// TIA Portal V20 export
FUNCTION "01 T1-A ARUNC Alarms" : Void   // FC1102, LAD
TITLE = ALARMS
{ S7_Optimized_Access := 'TRUE' }
// stored: AutoNumber false, IsIECCheckEnabled true, SetENOAutomatically false
   VAR_TEMP
      Trash : Bool;
   END_VAR
BEGIN

REGION Network 1: ============ ALARMS RESET ============
END_REGION

REGION Network 2: Alarms Reset
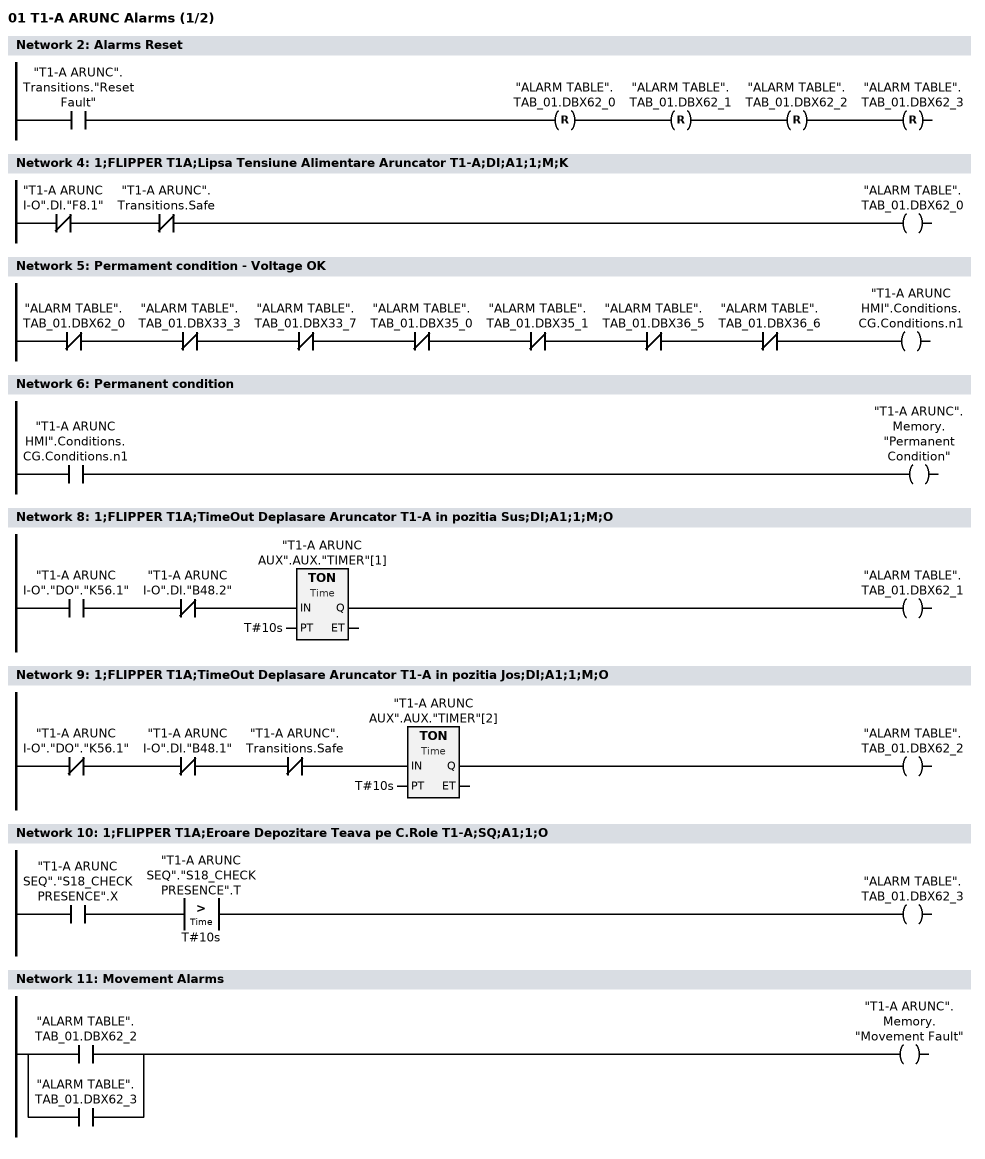
   RUNG wire#powerrail
      Contact( "T1-A ARUNC".Transitions."Reset Fault" )
      R_Coil( "ALARM TABLE".TAB_01.DBX62_0 )
      R_Coil( "ALARM TABLE".TAB_01.DBX62_1 )
      R_Coil( "ALARM TABLE".TAB_01.DBX62_2 )
      R_Coil( "ALARM TABLE".TAB_01.DBX62_3 )
   END_RUNG
   // the same network as SCL:
   IF "T1-A ARUNC".Transitions."Reset Fault" THEN
       "ALARM TABLE".TAB_01.DBX62_0 := FALSE;
       "ALARM TABLE".TAB_01.DBX62_1 := FALSE;
       "ALARM TABLE".TAB_01.DBX62_2 := FALSE;
       "ALARM TABLE".TAB_01.DBX62_3 := FALSE;
   END_IF;
END_REGION

REGION Network 3: ============ PERMANENT CONDITIONS ============
END_REGION

REGION Network 4: 1;FLIPPER T1A;Lipsa Tensiune Alimentare Aruncator T1-A;DI;A1;1;M;K
   RUNG wire#powerrail
      I_Contact( "T1-A ARUNC I-O".DI."F8.1" )
      I_Contact( "T1-A ARUNC".Transitions.Safe )
      Coil( "ALARM TABLE".TAB_01.DBX62_0 )
   END_RUNG
   // the same network as SCL:
   "ALARM TABLE".TAB_01.DBX62_0 := NOT "T1-A ARUNC I-O".DI."F8.1" AND NOT "T1-A ARUNC".Transitions.Safe;
END_REGION

REGION Network 5: Permament condition - Voltage OK
   RUNG wire#powerrail
      I_Contact( "ALARM TABLE".TAB_01.DBX62_0 )
      I_Contact( "ALARM TABLE".TAB_01.DBX33_3 )
      I_Contact( "ALARM TABLE".TAB_01.DBX33_7 )
      I_Contact( "ALARM TABLE".TAB_01.DBX35_0 )
      I_Contact( "ALARM TABLE".TAB_01.DBX35_1 )
      I_Contact( "ALARM TABLE".TAB_01.DBX36_5 )
      I_Contact( "ALARM TABLE".TAB_01.DBX36_6 )
      Coil( "T1-A ARUNC HMI".Conditions.CG.Conditions.n1 )
   END_RUNG
   // the same network as SCL:
   "T1-A ARUNC HMI".Conditions.CG.Conditions.n1 := NOT "ALARM TABLE".TAB_01.DBX62_0 AND NOT "ALARM TABLE".TAB_01.DBX33_3 AND NOT "ALARM TABLE".TAB_01.DBX33_7 AND NOT "ALARM TABLE".TAB_01.DBX35_0 AND NOT "ALARM TABLE".TAB_01.DBX35_1 AND NOT "ALARM TABLE".TAB_01.DBX36_5 AND NOT "ALARM TABLE".TAB_01.DBX36_6;
END_REGION

REGION Network 6: Permanent condition
   RUNG wire#powerrail
      Contact( "T1-A ARUNC HMI".Conditions.CG.Conditions.n1 )
      Coil( "T1-A ARUNC".Memory."Permanent Condition" )
   END_RUNG
   // the same network as SCL:
   "T1-A ARUNC".Memory."Permanent Condition" := "T1-A ARUNC HMI".Conditions.CG.Conditions.n1;
END_REGION

REGION Network 7: ======= MACHINE MOVEMENT CONTROL (SENSORS / ENCODERS / INTERLOCKS) =======
END_REGION

REGION Network 8: 1;FLIPPER T1A;TimeOut Deplasare Aruncator T1-A in pozitia Sus;DI;A1;1;M;O
   RUNG wire#powerrail
      Contact( "T1-A ARUNC I-O"."DO"."K56.1" )
      I_Contact( "T1-A ARUNC I-O".DI."B48.2" )
      { S7_Templates := "time_type := Time" } "T1-A ARUNC AUX".AUX."TIMER"[1].TON(pt := T#10s, et =>)
      Coil( "ALARM TABLE".TAB_01.DBX62_1 )
   END_RUNG
   // the same network as SCL:
   "T1-A ARUNC AUX".AUX."TIMER"[1].TON(IN := "T1-A ARUNC I-O"."DO"."K56.1" AND NOT "T1-A ARUNC I-O".DI."B48.2",
                           PT := T#10s);
   "ALARM TABLE".TAB_01.DBX62_1 := "T1-A ARUNC AUX".AUX."TIMER"[1].Q;
END_REGION

REGION Network 9: 1;FLIPPER T1A;TimeOut Deplasare Aruncator T1-A in pozitia Jos;DI;A1;1;M;O
   RUNG wire#powerrail
      I_Contact( "T1-A ARUNC I-O"."DO"."K56.1" )
      I_Contact( "T1-A ARUNC I-O".DI."B48.1" )
      I_Contact( "T1-A ARUNC".Transitions.Safe )
      { S7_Templates := "time_type := Time" } "T1-A ARUNC AUX".AUX."TIMER"[2].TON(pt := T#10s, et =>)
      Coil( "ALARM TABLE".TAB_01.DBX62_2 )
   END_RUNG
   // the same network as SCL:
   "T1-A ARUNC AUX".AUX."TIMER"[2].TON(IN := NOT "T1-A ARUNC I-O"."DO"."K56.1" AND NOT "T1-A ARUNC I-O".DI."B48.1" AND NOT "T1-A ARUNC".Transitions.Safe,
                           PT := T#10s);
   "ALARM TABLE".TAB_01.DBX62_2 := "T1-A ARUNC AUX".AUX."TIMER"[2].Q;
END_REGION

REGION Network 10: 1;FLIPPER T1A;Eroare Depozitare Teava pe C.Role T1-A;SQ;A1;1;O
   RUNG wire#powerrail
      Contact( "T1-A ARUNC SEQ"."S18_CHECK PRESENCE".X )
      { S7_Templates := "SrcType := Time" } GT_Contact(in1 := "T1-A ARUNC SEQ"."S18_CHECK PRESENCE".T, in2 := T#10s)
      Coil( "ALARM TABLE".TAB_01.DBX62_3 )
   END_RUNG
   // the same network as SCL:
   "ALARM TABLE".TAB_01.DBX62_3 := "T1-A ARUNC SEQ"."S18_CHECK PRESENCE".X AND ("T1-A ARUNC SEQ"."S18_CHECK PRESENCE".T > T#10s);
END_REGION

REGION Network 11: Movement Alarms
   RUNG wire#powerrail
      Contact( "ALARM TABLE".TAB_01.DBX62_2 )
      wire#w1
      Coil( "T1-A ARUNC".Memory."Movement Fault" )
   END_RUNG
   RUNG wire#powerrail
      Contact( "ALARM TABLE".TAB_01.DBX62_3 )
   END_RUNG wire#w1
   // the same network as SCL:
   "T1-A ARUNC".Memory."Movement Fault" := "ALARM TABLE".TAB_01.DBX62_2 OR "ALARM TABLE".TAB_01.DBX62_3;
END_REGION

REGION Network 12: ======= OTHER ALARMS =======
END_REGION

REGION Network 13: ======= FAULT =======
END_REGION

REGION Network 14: Fault Transition
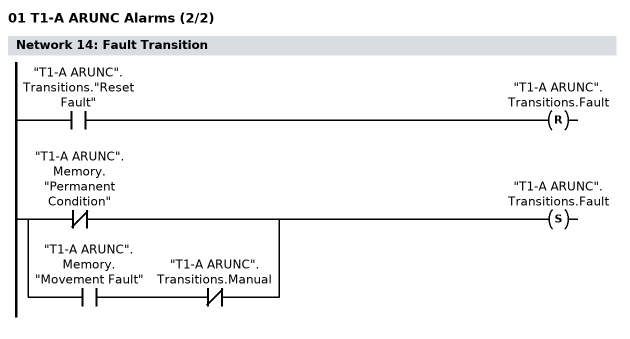
   RUNG wire#powerrail
      Contact( "T1-A ARUNC".Transitions."Reset Fault" )
      R_Coil( "T1-A ARUNC".Transitions.Fault )
   END_RUNG
   RUNG wire#powerrail
      I_Contact( "T1-A ARUNC".Memory."Permanent Condition" )
      wire#w1
      S_Coil( "T1-A ARUNC".Transitions.Fault )
   END_RUNG
   RUNG wire#powerrail
      Contact( "T1-A ARUNC".Memory."Movement Fault" )
      I_Contact( "T1-A ARUNC".Transitions.Manual )
   END_RUNG wire#w1
   // the same network as SCL:
   IF "T1-A ARUNC".Transitions."Reset Fault" THEN "T1-A ARUNC".Transitions.Fault := FALSE; END_IF;
   IF NOT "T1-A ARUNC".Memory."Permanent Condition" OR ("T1-A ARUNC".Memory."Movement Fault" AND NOT "T1-A ARUNC".Transitions.Manual) THEN
       "T1-A ARUNC".Transitions.Fault := TRUE;
   END_IF;
END_REGION
END_FUNCTION
